FUNCTION_BLOCK WORKER4TESTFB (* JADE WORKER *)
  (* Standard: 61499-1 *)
  (* Version 1.0, 2014-04-22, Ahmed, Fraunhofer IGD *)
  (* Compiler header: package fb.rt; *)
  (* Compiler Java Sun JDK 1.5.0 *)
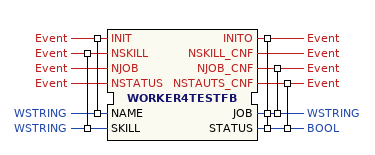
  EVENT_INPUT
    INIT WITH NAME; (* Normal Execution Request *)
    NSKILL WITH SKILL; (* Normal Execution Request *)
    NJOB;
    NSTATUS;
  END_EVENT
  EVENT_OUTPUT
    INITO WITH JOB, STATUS; (* Execution Confirmation *)
    NSKILL_CNF;
    NJOB_CNF WITH JOB;
    NSTAUTS_CNF WITH STATUS;
  END_EVENT
  VAR_INPUT
    NAME : WSTRING;
    SKILL : WSTRING;
  END_VAR
  VAR_OUTPUT
    JOB : WSTRING;
    STATUS : BOOL;
  END_VAR
END_FUNCTION_BLOCK
